FUNCTION_BLOCK DSTest
  (* Standard: 61499-2 *)
  (* Version 0.2, 2003-12-05, JHC, Rockwell Automation, Renamed from NEWCOMPFB. *)
  (* Version 0.1, 2002-01-08, JHC, Rockwell Automation, Added DLY FB as example. *)
  (* Version 0.0, 2000-05-27, JHC, Rockwell Automation *)
  (* Compiler header: package fb.rt.projects.DrillStation; *)
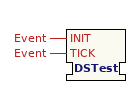
  EVENT_INPUT
    INIT; (* Initialization Request *)
    TICK; (* Normal Execution Request *)
  END_EVENT
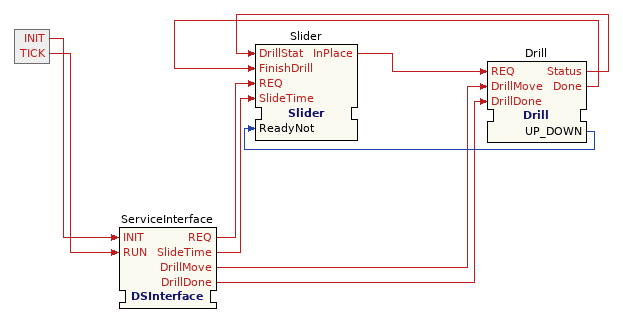
  FBS
    Drill : Drill;
    Slider : Slider;
    ServiceInterface : DSInterface;
  END_FBS
  EVENT_CONNECTIONS
    Drill.Status TO Slider.DrillStat;
    Drill.Done TO Slider.FinishDrill;
    Slider.InPlace TO Drill.REQ;
    ServiceInterface.REQ TO Slider.REQ;
    ServiceInterface.SlideTime TO Slider.SlideTime;
    ServiceInterface.DrillMove TO Drill.DrillMove;
    ServiceInterface.DrillDone TO Drill.DrillDone;
    INIT TO ServiceInterface.INIT;
    TICK TO ServiceInterface.RUN;
  END_CONNECTIONS
  DATA_CONNECTIONS
    Drill.UP_DOWN TO Slider.ReadyNot;
  END_CONNECTIONS
END_FUNCTION_BLOCK
